{library PUBLIC}
(* Station number type *)
TYPE StationType : INT(1..9);
END_TYPE

(* stored: Version 1.1.0.1, ProductVersion 3.1.4024.2
   EnumerationTextList StationType: Id {157cb296-1cb3-4d29-a4f4-0474d1be9029} *)
